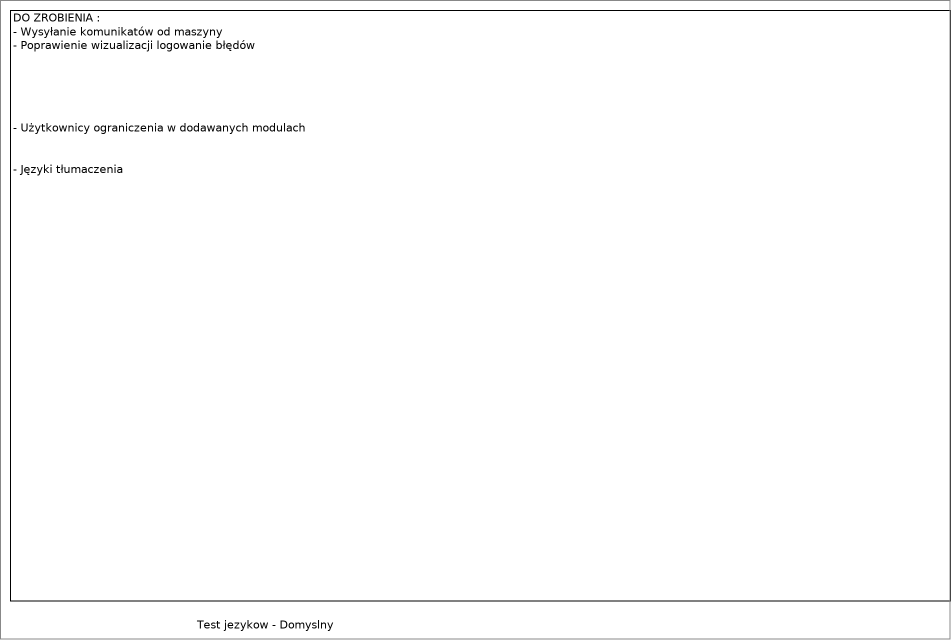
VISUALIZATION OknoGlowne  // 951x640
    Rectangle (10,10 941x591), "DO ZROBIENIA : - Wysyłanie komunikatów od maszyny - Poprawienie wizualizacji logowanie błędów - Użytkownicy ograniczenia w dodawanych modulach - Języki tłumaczenia"
    Label (50,610 431x30), "Test jezykow - Domyslny"
END_VISUALIZATION

(* stored: Version 1.1.0.1, ProductVersion 3.1.4024.11
   Visu OknoGlowne: Id {97ad123c-810a-4475-8dca-86386f36f6b7} *)
